FUNCTION_BLOCK FB_PMPSJsonTestHelper
(*
    Build a JSON document in memory from the input structs and publish
    it to the global PMPS doc (PMPS_GVL.BP_jsonDoc). Unlike
    FB_PMPSJsonTestHelperEx, this helper serializes the reactive
    temperature and pressure set points (nTempSP / nPressSP) into the
    reactive_temp / reactive_pressure members, so it is the helper to
    use for any device whose test reads a reactive-DB threshold.

    bNewDoc selects the document mode: TRUE creates a fresh root
    document (first device in the seeding chain); FALSE appends this
    device to the existing PMPS_GVL.BP_jsonDoc, so several helpers can
    accumulate into one multi-device document.
*)
VAR_IN_OUT
    astBeamParams: ARRAY[*] OF ST_DbStateParams;
END_VAR
VAR_INPUT
    bExecute: BOOL;
    sDevName: STRING;
    bNewDoc: BOOL;
END_VAR
VAR_OUTPUT
END_VAR
VAR
    rtExec: R_TRIG;
    jsonRoot: SJsonValue;
    jsonDevice: SJsonValue;
    ajsonState: ARRAY[0..GeneralConstants.MAX_STATES] OF SJsonValue;
    fbJson: FB_JsonDomParser;

    nIter: DINT;
    nId: DINT;

    aseVRange: ARRAY[0..GeneralConstants.MAX_STATES] OF STRING;
    asRate: ARRAY[0..GeneralConstants.MAX_STATES] OF STRING;
    asBCRange: ARRAY[0..GeneralConstants.MAX_STATES] OF STRING;
    asTran: ARRAY[0..GeneralConstants.MAX_STATES] OF STRING;

    sTemp: STRING;
    sPress: STRING;
END_VAR


rtExec(CLK:=bExecute);
IF NOT rtExec.Q THEN
    RETURN;
END_IF

IF bNewDoc THEN
    jsonRoot := fbJson.NewDocument();
ELSE
    jsonRoot := PMPS_GVL.BP_jsonDoc;
END_IF
jsonDevice := fbJson.AddObjectMember(jsonRoot, sDevName);
FOR nIter := LOWER_BOUND(astBeamParams, 1) TO UPPER_BOUND(astBeamParams, 1) DO
    ajsonState[nIter] := fbJson.AddObjectMember(jsonDevice, astBeamParams[nIter].sPmpsState);

    // Prefer the seeded assertion ID as the DB 'id' so it is unique and
    // meaningful; fall back to a running counter when a state leaves
    // nRequestAssertionID unset, so 'id' is never 0.
    nId := nId + 1;
    IF astBeamParams[nIter].nRequestAssertionID <> 0 THEN
        fbJson.AddIntMember(
            v:=ajsonState[nIter],
            member:='id',
            value:=UDINT_TO_DINT(astBeamParams[nIter].nRequestAssertionID),
        );
    ELSE
        fbJson.AddIntMember(
            v:=ajsonState[nIter],
            member:='id',
            value:=nId,
        );
    END_IF
    fbJson.AddStringMember(
        v:=ajsonState[nIter],
        member:='beamline',
        value:='tst',
    );
    aseVRange[nIter] := bitmaskToString(astBeamParams[nIter].stBeamParams.neVRange, 32);
    fbJson.AddStringMember(
        v:=ajsonState[nIter],
        member:='neVRange',
        value:=aseVRange[nIter],
    );
    asRate[nIter] := UDINT_TO_STRING(astBeamParams[nIter].stBeamParams.nRate);
    fbJson.AddStringMember(
        v:=ajsonState[nIter],
        member:='nRate',
        value:=asRate[nIter],
    );
    fbJson.AddStringMember(
        v:=ajsonState[nIter],
        member:='ap_ygap',
        value:='',
    );
    fbJson.AddStringMember(
        v:=ajsonState[nIter],
        member:='ap_xgap',
        value:='',
    );
    fbJson.AddStringMember(
        v:=ajsonState[nIter],
        member:='damage_limit',
        value:='',
    );
    fbJson.AddStringMember(
        v:=ajsonState[nIter],
        member:='notes',
        value:='',
    );
    sTemp := TO_STRING(astBeamParams[nIter].stReactiveParams.nTempSP);
    fbJson.AddStringMember(
        v:=ajsonState[nIter],
        member:='reactive_temp',
        value:=sTemp,
    );
    sPress := TO_STRING(astBeamParams[nIter].stReactiveParams.nPressSP);
    fbJson.AddStringMember(
        v:=ajsonState[nIter],
        member:='reactive_pressure',
        value:=sPress,
    );
    asBCRange[nIter] := bitmaskToString(astBeamParams[nIter].stBeamParams.nBCRange, 15);
    fbJson.AddStringMember(
        v:=ajsonState[nIter],
        member:='nBeamClassRange',
        value:=asBCRange[nIter],
    );
    fbJson.AddStringMember(
        v:=ajsonState[nIter],
        member:='name',
        value:=astBeamParams[nIter].sPmpsState,
    );
    asTran[nIter] := REAL_TO_STRING(astBeamParams[nIter].stBeamParams.nTran);
    fbJson.AddStringMember(
        v:=ajsonState[nIter],
        member:='nTran',
        value:=asTran[nIter],
    );
    fbJson.AddStringMember(
        v:=ajsonState[nIter],
        member:='ap_name',
        value:='None',
    );
    fbJson.AddStringMember(
        v:=ajsonState[nIter],
        member:='ap_ycenter',
        value:='',
    );
    fbJson.AddStringMember(
        v:=ajsonState[nIter],
        member:='ap_xcenter',
        value:='',
    );
    fbJson.AddStringMember(
        v:=ajsonState[nIter],
        member:='pulse_energy',
        value:='',
    );
    fbJson.AddBoolMember(
        v:=ajsonState[nIter],
        member:='special',
        value:=FALSE,
    );
END_FOR

PMPS_GVL.BP_jsonDoc := jsonRoot;

METHOD bitmaskToString : STRING
VAR_INPUT
    nBitmask: DWORD;
    nBits: UINT;
END_VAR
VAR
    nIter: UINT;
END_VAR

bitmaskToString := '';
FOR nIter := 1 TO nBits DO
    bitmaskToString := CONCAT(DWORD_TO_STRING(SHR(nBitmask, nIter - 1) AND 1), bitmaskToString);
END_FOR
END_METHOD

END_FUNCTION_BLOCK

(* stored: Version 1.1.0.1
   POU FB_PMPSJsonTestHelper: Id {dc71dc31-2d0b-4062-b2d3-b26324b3473f}, SpecialFunc None
   Method bitmaskToString: Id {a74cbfbf-040a-4efc-a4a9-225eb526d334} *)
